// TIA Portal project "VtSys_V13_SP1" (V13)

(* hardware
DEVICE "S7300/ET200M-Station_1"  S7-300 station
   slot 0: "Profilschiene_0"  Rail  6ES7 390-1***0-0AA0
   slot 1: "PS 307 5A_1"  PS 307 5A  6ES7 307-1EA00-0AA0
   slot 2: "S7-300 PLC"  CPU 314C-2 PN/DP  6ES7 314-6EH04-0AB0  V3.3
      slot 2: "PROFINET-Schnittstelle_1"  PN-IO
         slot 1: "Port_1"  Port
         slot 2: "Port_2"  Port
      slot 5: "DI 24/DO 16_1"  DI24/DO16
      slot 6: "AI 5/AO 2_1"  AI5/AO2
      slot 7: "Zählen_1"  Counter
      slot 8: "Positionieren_1"  Positioning
   slot 4: "CP 343-2_1"  CP 343-2  6GK7 343-2AH01-0XA0  V3.1
*)

// ===== PLC "S7-300 PLC"  CPU 314C-2 PN/DP =====

VAR_GLOBAL   // PLC tag table "Standard-Variablentabelle"
   "Mx_Clock10Hz" AT %M100.0 : Bool;   // CPU clock memory-flag 0: T=0,1 s/ f=10 Hz
   "Mx_Clock5Hz" AT %M100.1 : Bool;   // CPU clock memory-flag 1: T=0,2 s/ f=5 Hz
   "Mx_Clock2.5Hz" AT %M100.2 : Bool;   // CPU clock memory-flag 2: T=0,4 s/ f=2,5 Hz
   "Mx_Clock2Hz" AT %M100.3 : Bool;   // CPU clock memory-flag 3: T=0,5 s/ f=2 Hz
   "Mx_Clock1.25Hz" AT %M100.4 : Bool;   // CPU-Taktmerker-Bit 4: f=10Hz / T=0.8s
   "Mx_Clock1Hz" AT %M100.5 : Bool;   // CPU clock memory-flag 4: T=0,8 s/ f=1,25 Hz
   "Mx_Clock0.625Hz" AT %M100.6 : Bool;   // CPU clock memory-flag 6: T=1,6 s/ f=0,625 Hz
   "Mx_Clock0.5Hz" AT %M100.7 : Bool;   // CPU clock memory-flag 7: T=2 s/ f=0,5 Hz
   "Qx_P_RD" AT %Q124.0 : Bool;   // Traffic light red
   "Qx_P_YE" AT %Q124.1 : Bool;   // Traffic light yellow
   "Qx_P_GN" AT %Q124.2 : Bool;   // Traffic light green
   "Qx_Q1 (P1)" AT %Q125.0 : Bool;   // Fan motor 1 (main contactor and signal lamp)
   "Qx_Q2 (P2)" AT %Q125.1 : Bool;   // Fan motor 2 (main contactor and signal lamp)
   "Qx_Q3 (P3)" AT %Q125.2 : Bool;   // Fan motor 3 (main contactor and signal lamp)
   "Qx_Q4 (P4)" AT %Q125.3 : Bool;   // Fan motor 4 (main contactor and signal lamp)
   "Mx_Lock-C" AT %M20.3 : Bool;   // The counter must be locked as soon as the underground parking is full
   "Mx_PEdgeFlag_Step1" AT %M20.2 : Bool;   // Positive edge flag is activated when step 1 is activated
   "Mx_StartingFlag" AT %M20.0 : Bool;   // starting flag to activate the sequence (step 1)
   "Mx_Step1" AT %M10.0 : Bool;   // Grafcet G1, step-flag 1
   "Mx_Step2" AT %M10.1 : Bool;   // Grafcet G1, step-flag 2
   "Mx_Step20" AT %M10.2 : Bool;   // Grafcet G20, step-flag 20
   "Mx_Step30" AT %M10.3 : Bool;   // Grafcet G30, step-flag 30
   "Ix_S0" AT %I124.0 : Bool;   // Fan motors M1 to M4 off (NC)
   "Ix_F1_(S1)" AT %I124.1 : Bool;   // Overload relay F1, motor 1 (NC)
   "Ix_F2_(S2)" AT %I124.2 : Bool;   // Overload relay F2, motor 2 (NC)
   "Ix_F3_(S3)" AT %I124.3 : Bool;   // Overload relay F3, motor 3 (NC)
   "Ix_F4_(S4)" AT %I124.4 : Bool;   // Overload relay F4, motor 4 (NC)
   "Ix_S5" AT %I124.5 : Bool;   // Fan motors M1 to M4 on
   "Ix_B1" AT %I124.6 : Bool;   // Sensor to detect incoming vehicles
   "Ix_B2" AT %I124.7 : Bool;   // Sensor to detect outgoing vehicles
   "Ix_S6_(Reset)" AT %I125.0 : Bool;   // Reset vehicle counter
   "Mb_StepFlag" AT %MB10 : Byte;   // Step-flag byte 10
   "Mw_CV_INT" AT %MW32 : Int;   // Count value in the format INTEGER
   "Mw_CV_WORD" AT %MW30 : Word;   // Count value in the format WORD
   "C_Vehicle-C" AT %C1 : Counter;   // Counter to count the number of vehicles
END_VAR

DATA_BLOCK "Fan 1"   // DB11
{ S7_Optimized_Access := 'FALSE' }
VERSION : 0.1
// stored: InstanceOfName Grafcet G1X
"Grafcet G1X"
BEGIN
END_DATA_BLOCK

DATA_BLOCK "Fan 2"   // DB12
{ S7_Optimized_Access := 'FALSE' }
VERSION : 0.1
// stored: InstanceOfName Grafcet G1X
"Grafcet G1X"
BEGIN
END_DATA_BLOCK

DATA_BLOCK "Fan 3"   // DB13
{ S7_Optimized_Access := 'FALSE' }
VERSION : 0.1
// stored: InstanceOfName Grafcet G1X
"Grafcet G1X"
BEGIN
END_DATA_BLOCK

DATA_BLOCK "Fan 4"   // DB14
{ S7_Optimized_Access := 'FALSE' }
VERSION : 0.1
// stored: InstanceOfName Grafcet G1X
"Grafcet G1X"
BEGIN
END_DATA_BLOCK

FUNCTION_BLOCK "Grafcet G1X"   // FB10, FBD
TITLE = Function diagram G1X (Partial GRAFCET "Fan X")
{ S7_Optimized_Access := 'FALSE' }
VERSION : 0.1
// Fan control
   VAR_TEMP   // added for the SCL form of the ladder/FBD networks
      _w1 : Bool;
      _w2 : Bool;
   END_VAR
BEGIN

REGION Network 1: Step 1Xa
   // A dominant setting self-latching relay must be used! The step 1Xa cannot be set if step 1Xb is already active.
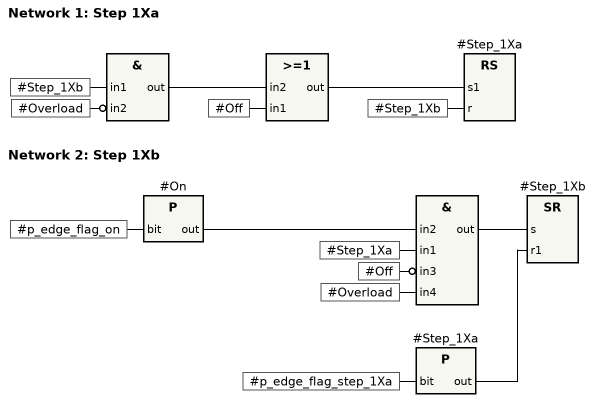
   IF #Step_1Xb THEN
       #Step_1Xa := FALSE;   // RS flip-flop
   END_IF;
   IF (#Step_1Xb AND NOT #Overload) OR #Off THEN #Step_1Xa := TRUE; END_IF;
END_REGION

REGION Network 2: Step 1Xb
   #_w1 := #On AND NOT #p_edge_flag_on;   // rising edge of #On
   #p_edge_flag_on := #On;
   #_w2 := #Step_1Xa AND NOT #p_edge_flag_step_1Xa;   // rising edge of #Step_1Xa
   #p_edge_flag_step_1Xa := #Step_1Xa;
   IF #_w1 AND #Step_1Xa AND NOT #Off AND #Overload THEN
       #Step_1Xb := TRUE;   // SR flip-flop
   END_IF;
   IF #_w2 THEN #Step_1Xb := FALSE; END_IF;
END_REGION
END_FUNCTION_BLOCK

FUNCTION "Grafcet G1" : Void   // FC1, FBD
TITLE = Function diagram G1 (Partial GRAFCET "main switch")
{ S7_Optimized_Access := 'FALSE' }
VERSION : 0.1
   VAR_TEMP   // added for the SCL form of the ladder/FBD networks
      _w1 : Bool;
   END_VAR
BEGIN

REGION Network 1: Step 1
   // A dominant setting self-latching relay must be used! The step 1 cannot be set if step 2 is already active.
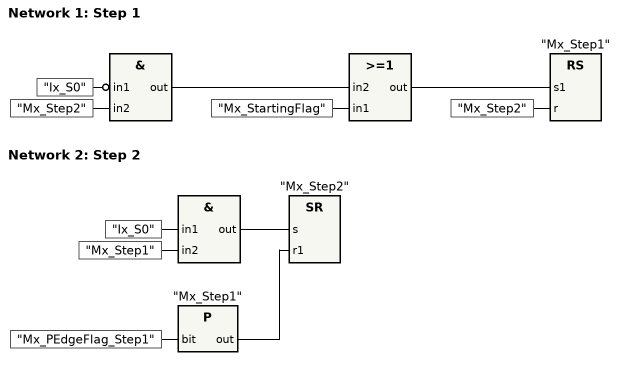
   IF "Mx_Step2" THEN
       "Mx_Step1" := FALSE;   // RS flip-flop
   END_IF;
   IF (NOT "Ix_S0" AND "Mx_Step2") OR "Mx_StartingFlag" THEN "Mx_Step1" := TRUE; END_IF;
END_REGION

REGION Network 2: Step 2
   #_w1 := "Mx_Step1" AND NOT "Mx_PEdgeFlag_Step1";   // rising edge of "Mx_Step1"
   "Mx_PEdgeFlag_Step1" := "Mx_Step1";
   IF "Ix_S0" AND "Mx_Step1" THEN
       "Mx_Step2" := TRUE;   // SR flip-flop
   END_IF;
   IF #_w1 THEN "Mx_Step2" := FALSE; END_IF;
END_REGION
END_FUNCTION

FUNCTION "Actions" : Void   // FC2, FBD
TITLE = Execute the actions
{ S7_Optimized_Access := 'FALSE' }
VERSION : 0.1
BEGIN

REGION Network 1: Control fan 1
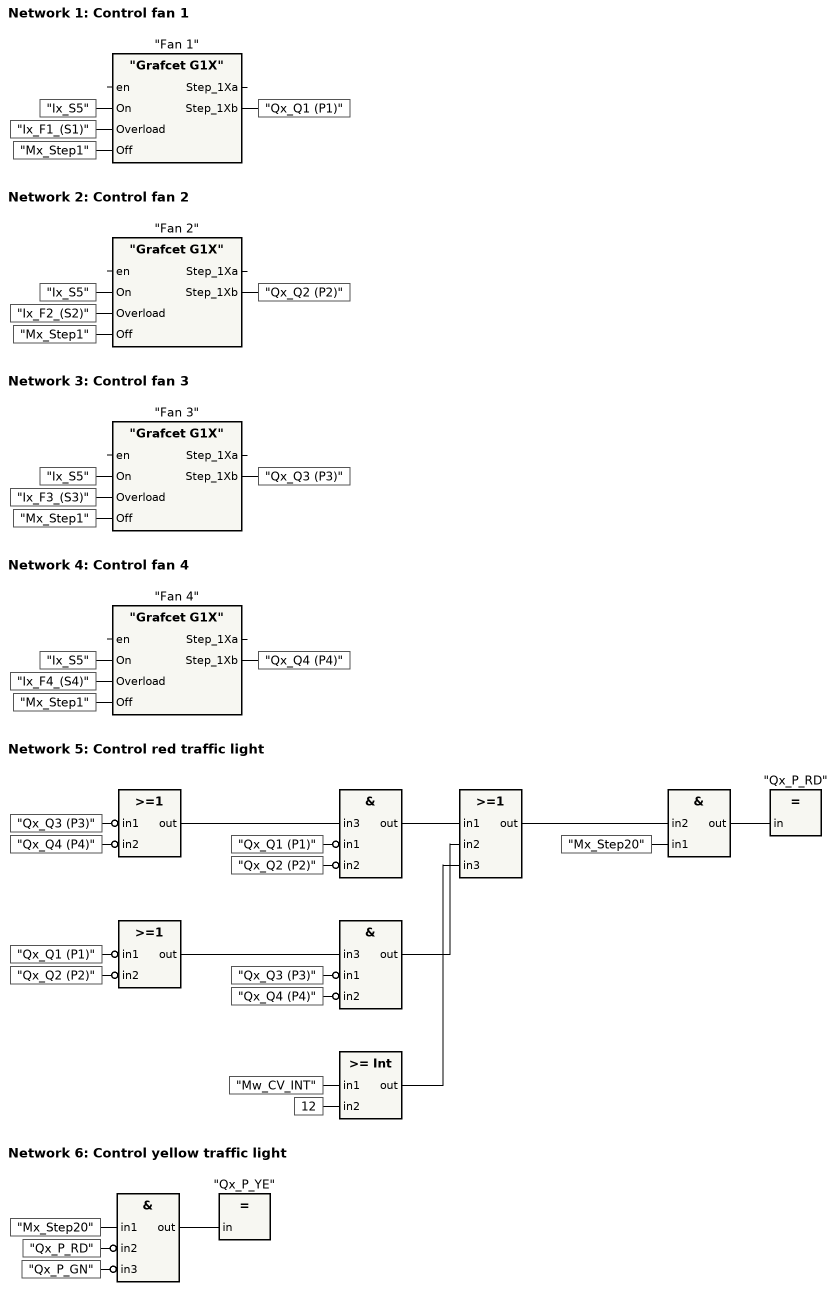
   "Fan 1"(On := "Ix_S5", Overload := "Ix_F1_(S1)", Off := "Mx_Step1", Step_1Xb => "Qx_Q1 (P1)");   // "Grafcet G1X"
END_REGION

REGION Network 2: Control fan 2
   "Fan 2"(On := "Ix_S5", Overload := "Ix_F2_(S2)", Off := "Mx_Step1", Step_1Xb => "Qx_Q2 (P2)");   // "Grafcet G1X"
END_REGION

REGION Network 3: Control fan 3
   "Fan 3"(On := "Ix_S5", Overload := "Ix_F3_(S3)", Off := "Mx_Step1", Step_1Xb => "Qx_Q3 (P3)");   // "Grafcet G1X"
END_REGION

REGION Network 4: Control fan 4
   "Fan 4"(On := "Ix_S5", Overload := "Ix_F4_(S4)", Off := "Mx_Step1", Step_1Xb => "Qx_Q4 (P4)");   // "Grafcet G1X"
END_REGION

REGION Network 5: Control red traffic light
   // The traffic light works only if step 20 is active.
   "Qx_P_RD" := (((NOT "Qx_Q3 (P3)" OR NOT "Qx_Q4 (P4)") AND NOT "Qx_Q1 (P1)" AND NOT "Qx_Q2 (P2)") OR ((NOT "Qx_Q1 (P1)" OR NOT "Qx_Q2 (P2)") AND NOT "Qx_Q3 (P3)" AND NOT "Qx_Q4 (P4)") OR ("Mw_CV_INT" >= 12)) AND "Mx_Step20";
END_REGION

REGION Network 6: Control yellow traffic light
   // The traffic light works only if step 20 is active.
   "Qx_P_YE" := "Mx_Step20" AND NOT "Qx_P_RD" AND NOT "Qx_P_GN";
END_REGION

REGION Network 7: Control green traffic light
   // The traffic light works only if step 20 is active. As soon as 12 vehicles are in the underground parking, only the red lamp must light. The green lamp may not light any longer, even if this were possible, due to the number of fans in operation. Therefore the green lamp must additionally be locked with the red lamp.
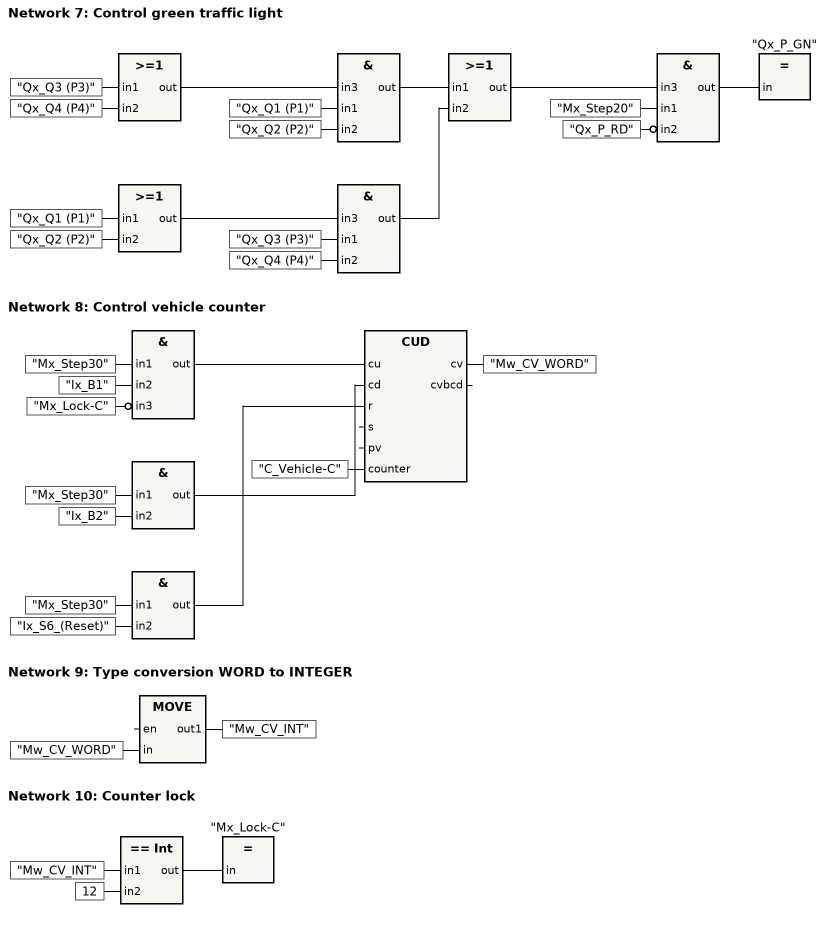
   "Qx_P_GN" := ((("Qx_Q3 (P3)" OR "Qx_Q4 (P4)") AND "Qx_Q1 (P1)" AND "Qx_Q2 (P2)") OR (("Qx_Q1 (P1)" OR "Qx_Q2 (P2)") AND "Qx_Q3 (P3)" AND "Qx_Q4 (P4)")) AND "Mx_Step20" AND NOT "Qx_P_RD";
END_REGION

REGION Network 8: Control vehicle counter
   // The vehicle counter (up counter, down counter and reset) works only if step 30 is active.
   // no SCL statement known for Cud: written as a call
   Cud(cu := "Mx_Step30" AND "Ix_B1" AND NOT "Mx_Lock-C",
       cd := "Mx_Step30" AND "Ix_B2",
       r := "Mx_Step30" AND "Ix_S6_(Reset)",
       "counter" := "C_Vehicle-C",
       cv => "Mw_CV_WORD");
END_REGION

REGION Network 9: Type conversion WORD to INTEGER
   // The counter block (see network 8) expects at the output CV_BCD a value of the type WORD and the compare block "CMP" (see network 5) expects at the input IN a value of the type INTEGER. With the help of the "MOVE" operation (see below) 
   // one can do a type conversion from WORD to INTEGER.
   "Mw_CV_INT" := "Mw_CV_WORD";
END_REGION

REGION Network 10: Counter lock
   // Flag M20.3 is used for locking the counter (see network 8).
   "Mx_Lock-C" := "Mw_CV_INT" = 12;
END_REGION
END_FUNCTION

FUNCTION "Grafcet G20" : Void   // FC20, FBD
TITLE = Function diagram G20 (Partial GRAFCET "traffic light")
{ S7_Optimized_Access := 'FALSE' }
VERSION : 0.1
BEGIN

REGION Network 1: Step 20
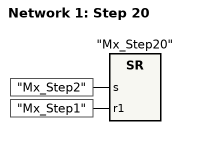
   IF "Mx_Step2" THEN
       "Mx_Step20" := TRUE;   // SR flip-flop
   END_IF;
   IF "Mx_Step1" THEN "Mx_Step20" := FALSE; END_IF;
END_REGION
END_FUNCTION

FUNCTION "Grafcet G30" : Void   // FC30, FBD
TITLE = Function diagram G30 (Partial GRAFCET "vehicle counter")
{ S7_Optimized_Access := 'FALSE' }
VERSION : 0.1
BEGIN

REGION Network 1: Step 30
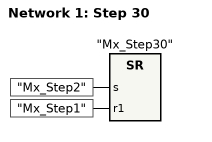
   IF "Mx_Step2" THEN
       "Mx_Step30" := TRUE;   // SR flip-flop
   END_IF;
   IF "Mx_Step1" THEN "Mx_Step30" := FALSE; END_IF;
END_REGION
END_FUNCTION

ORGANIZATION_BLOCK "Main"   // OB1, FBD
TITLE = "Main Program Sweep (Cycle)"
{ S7_Optimized_Access := 'FALSE' }
VERSION : 0.1
BEGIN

REGION Network 1: Call the function diagram block G1 ("main switch")
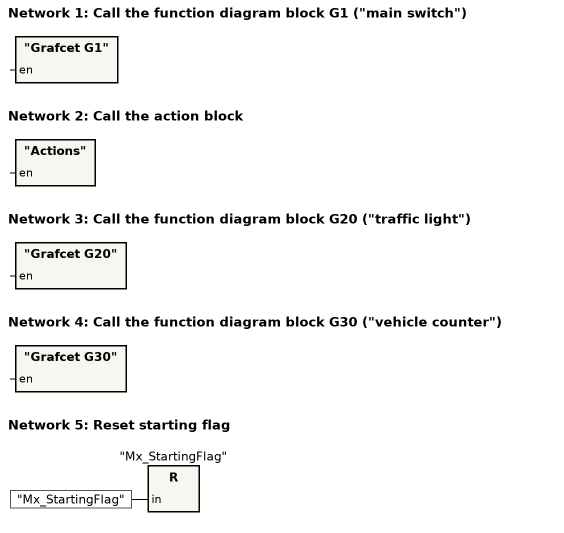
   "Grafcet G1"();
END_REGION

REGION Network 2: Call the action block
   "Actions"();
END_REGION

REGION Network 3: Call the function diagram block G20 ("traffic light")
   "Grafcet G20"();
END_REGION

REGION Network 4: Call the function diagram block G30 ("vehicle counter")
   "Grafcet G30"();
END_REGION

REGION Network 5: Reset starting flag
   IF "Mx_StartingFlag" THEN "Mx_StartingFlag" := FALSE; END_IF;
END_REGION
END_ORGANIZATION_BLOCK

ORGANIZATION_BLOCK "COMPLETE RESTART"   // OB100, FBD
TITLE = "Complete Restart"
{ S7_Optimized_Access := 'FALSE' }
VERSION : 0.1
BEGIN

REGION Network 1: Reset flag byte number 10
   // With the instruction "MOVE", all bits of memory flag byte number 10 will be overwritten with the value 0! Thus it is guaranteed that all steps are deactivated when the status of the PLC changes from RUN to STOP and back to 
   // RUN. Otherwise the plant will go back to the previous status without activating any pushbuttons.
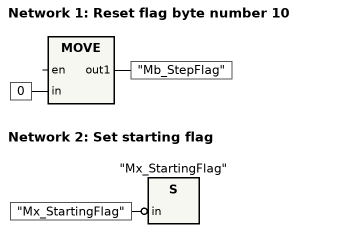
   "Mb_StepFlag" := 0;
END_REGION

REGION Network 2: Set starting flag
   IF NOT "Mx_StartingFlag" THEN "Mx_StartingFlag" := TRUE; END_IF;
END_REGION
END_ORGANIZATION_BLOCK